Staubli VAL3: Form_Main.pgx

public program Form_Main(string& x_sBottomList[])
  local num l_nIndex
begin
  //欢迎界面，显示日期和时间
 userPage()
cls()
 call Control_PanelMd("下位机处在主界面")



//     for l_nIndex=0 to min(7,size(x_sBottomList)-1)
//    gotoxy(1+l_nIndex*5,13)
//    if size(x_sBottomList)>l_nIndex and x_sBottomList[l_nIndex]!=""
//      put(x_sBottomList[l_nIndex])
//    endIf
//    endFor
 call Control_Bottom(x_sBottomList)
end
